FUNCTION CheckDivByte : BYTE
VAR_INPUT
	divisor			 	: BYTE;
END_VAR
VAR
END_VAR

IF divisor = 0 THEN
	CheckByteZeroDiv_ErrCnt := CheckByteZeroDiv_ErrCnt + 1;
	CheckDivByte := 1;
ELSE
	CheckDivByte := divisor;
END_IF

END_FUNCTION

(* stored: Version 1.1.0.1, ProductVersion 3.1.4024.12
   POU CheckDivByte: Id {78bd2019-7a26-444f-bd20-4f050ebbf05f}, SpecialFunc CheckDivInt32 *)
